# EPICS substitutions: iocs/diagnosticsTest/diagnosticsTestApp/Db/diagnostics_test.substitutions
# EtherCAT Master

file $(ETHERCAT)/db/MASTER.template
{
pattern {       DEVICE , PORT    , SCAN       }
        { rjq35657:sim , MASTER0 , "I/O Intr" }
}

file $(ETHERCAT)/db/EL3104.template
{
pattern {   DEVICE    , PORT ,     SCAN   }
        { RJQ35657:AI1,  AI1 , ".1 second"}
        { RJQ35657:AI2,  AI2 , ".1 second"}
}

file $(ETHERCAT)/db/gadc.template
{
pattern { DEVICE, CHANNEL, PORT, SAMPLES, SCAN , INTSCAN}
{RJQ35657-AMP-01:CHANNELA, 1, AI1, 1000, "I/O Intr", "Passive" }
{RJQ35657-AMP-01:CHANNELB, 2, AI1, 1000, "I/O Intr", "Passive" }
{RJQ35657-AMP-01:CHANNELC, 1, AI2, 1000, "I/O Intr", "Passive" }
{RJQ35657-AMP-01:CHANNELD, 2, AI2, 1000, "I/O Intr", "Passive" }

}
